{attribute 'qualified_only'}
{attribute 'strict'}
{attribute 'to_string'}
TYPE LogLevel :
(
	Debug := 0,
	Information,
	Warning,
	Error,
	Fatal
);
END_TYPE

(* stored: Version 1.1.0.1
   DUT LogLevel: Id {b22d3fef-91d4-49da-9c4a-eb3786bf2a9d} *)
